FUNCTION_BLOCK FB_Switch_Test EXTENDS TcUnit.FB_TestSuite
VAR
	_fbDevice 		: FB_Switch;
	_nExpected 		: BYTE;
	_nResult 		: BYTE;
END_VAR

TEST('Set nControl');
_nExpected := 255;
_fbDevice.nControl := _nExpected;
_fbDevice();
_nResult := _fbDevice.GetControl();

AssertEquals(Expected := _nExpected,
             Actual := _nResult,
             Message := 'Value is not correct');	
TEST_FINISHED();

TEST('Get nStatus');
_nExpected := 255;
_fbDevice.SetStatus(_nExpected);
_fbDevice();
_nResult := _fbDevice.nStatus;

AssertEquals(Expected := _nExpected,
             Actual := _nResult,
             Message := 'Value is not correct');	
TEST_FINISHED();

END_FUNCTION_BLOCK

(* stored: Version 1.1.0.1, ProductVersion 3.1.4024.12
   POU FB_Switch_Test: Id {a6702d73-a8b2-0087-133f-37c267a44a11}, SpecialFunc None *)
